TYPE tyRampdata_toDb :
STRUCT
	iRampStepOutput : INT ;
	tRampStepTime : TIME ; 
	
END_STRUCT
END_TYPE

(* stored: Version 1.1.0.1
   DUT tyRampdata_toDb: Id {b990cd32-65e7-47d7-8e26-3319205349eb} *)
